% RSLogix 500 project SERVO_PROJECT.RSS, saved by version 8.30.00.16 %
PROJECT "UNTITLED"    % processor: Bul.1763 MicroLogix 1100 Series B %

PROGRAM FILES
  LAD 2 "MAIN"  4 rungs
  LAD 3 "INPUT"  7 rungs
  LAD 4 "OUTPUT"  2 rungs
  LAD 5 "CONTROL"  29 rungs

DATA FILES
  O0 OUTPUT  4 elements
  I1 INPUT  6 elements
  S2 STATUS  66 elements
  B3 BINARY  4 elements
  T4 TIMER  3 elements
  C5 COUNTER  1 elements
  R6 CONTROL  1 elements
  N7 INTEGER  4 elements
  F8 FLOAT  1 elements

LADDER 2 "MAIN"
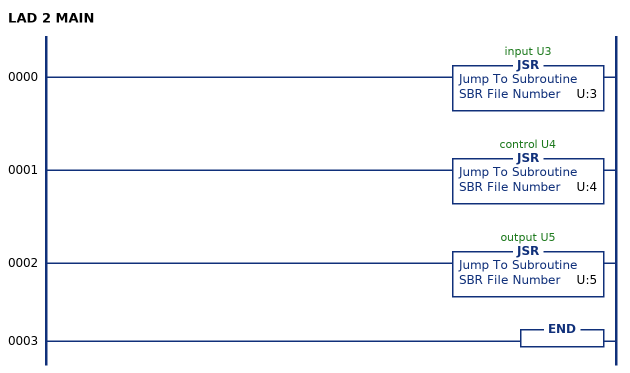
% Rung: 0 %
SOR JSR U:3 EOR
%   U:3  U3  "input" %
% Rung: 1 %
SOR JSR U:4 EOR
%   U:4  U4  "control" %
% Rung: 2 %
SOR JSR U:5 EOR
%   U:5  U5  "output" %
% Rung: 3 %
SOR END EOR

LADDER 3 "INPUT"
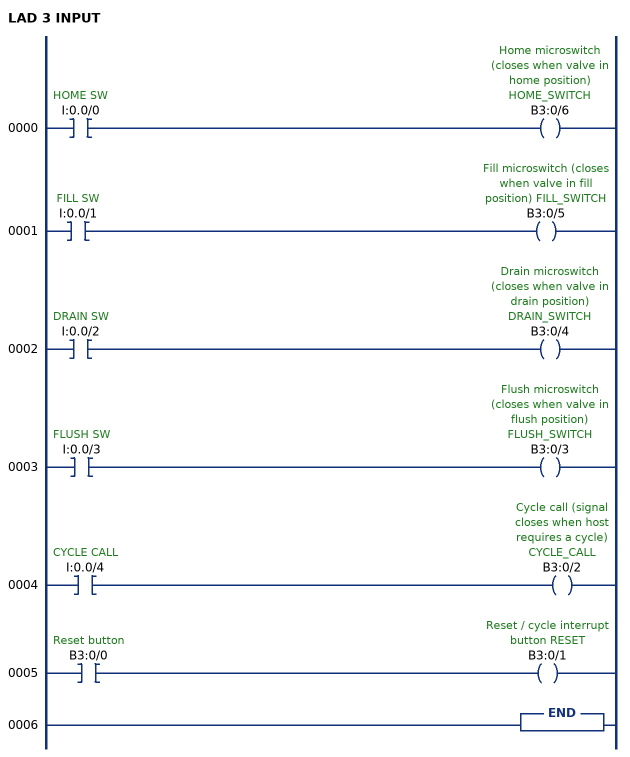
% Rung: 0 %
SOR XIC I:0.0/0 OTE B3:0/6 EOR
%   I:0.0/0  "HOME SW" %
%   B3:0/6  HOME_SWITCH  "Home microswitch (closes when valve in home position)" %
% Rung: 1 %
SOR XIC I:0.0/1 OTE B3:0/5 EOR
%   I:0.0/1  "FILL SW" %
%   B3:0/5  FILL_SWITCH  "Fill microswitch (closes when valve in fill position)" %
% Rung: 2 %
SOR XIC I:0.0/2 OTE B3:0/4 EOR
%   I:0.0/2  "DRAIN SW" %
%   B3:0/4  DRAIN_SWITCH  "Drain microswitch (closes when valve in drain position)" %
% Rung: 3 %
SOR XIC I:0.0/3 OTE B3:0/3 EOR
%   I:0.0/3  "FLUSH SW" %
%   B3:0/3  FLUSH_SWITCH  "Flush microswitch (closes when valve in flush position)" %
% Rung: 4 %
SOR XIC I:0.0/4 OTE B3:0/2 EOR
%   I:0.0/4  "CYCLE CALL" %
%   B3:0/2  CYCLE_CALL  "Cycle call (signal closes when host requires a cycle)" %
% Rung: 5 %
SOR XIC B3:0/0 OTE B3:0/1 EOR
%   B3:0/0  "Reset button" %
%   B3:0/1  RESET  "Reset / cycle interrupt button" %
% Rung: 6 %
SOR END EOR

LADDER 4 "OUTPUT"
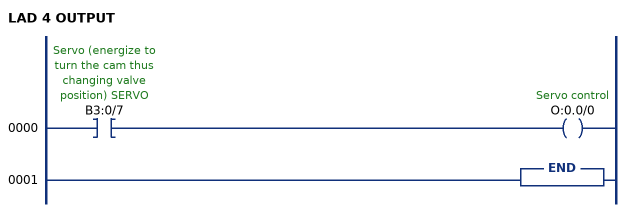
% Rung: 0 %
SOR XIC B3:0/7 OTE O:0.0/0 EOR
%   B3:0/7  SERVO  "Servo (energize to turn the cam thus changing valve position)" %
%   O:0.0/0  "Servo control" %
% Rung: 1 %
SOR END EOR

LADDER 5 "CONTROL"
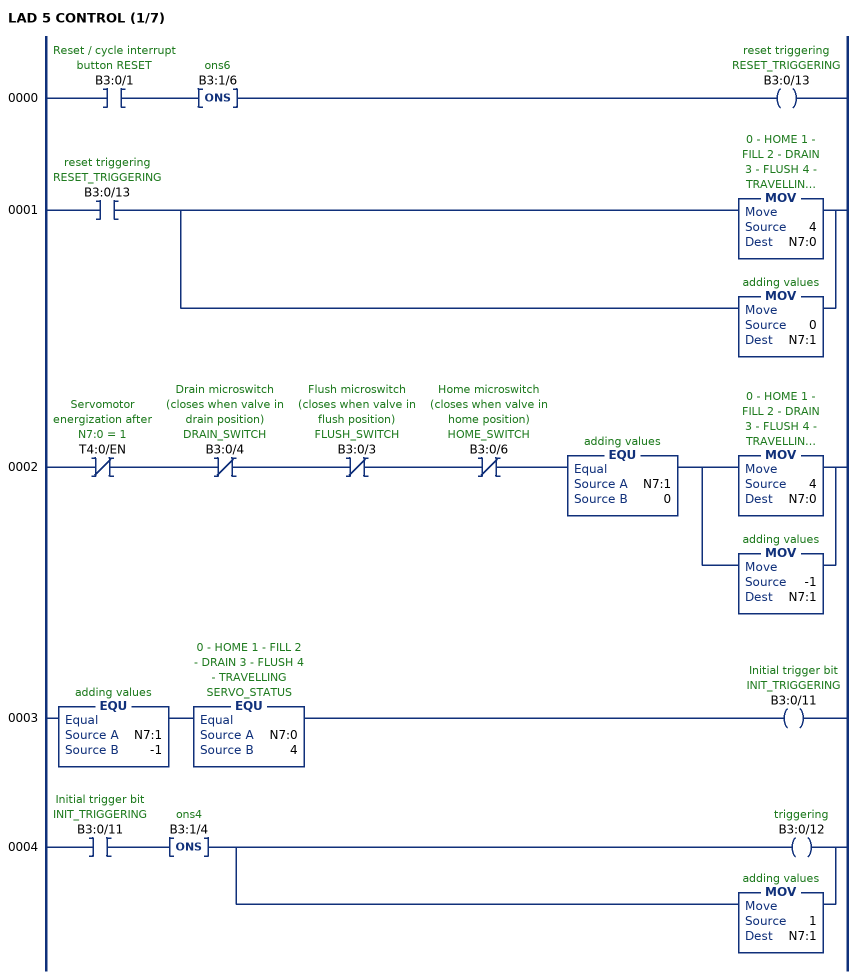
% Rung: 0 %
SOR XIC B3:0/1 ONS B3:1/6 OTE B3:0/13 EOR
%   B3:0/1  RESET  "Reset / cycle interrupt button" %
%   B3:1/6  "ons6" %
%   B3:0/13  RESET_TRIGGERING  "reset triggering" %
% Rung: 1 %
SOR XIC B3:0/13 BST MOV 4 N7:0 NXB MOV 0 N7:1 BND EOR
%   B3:0/13  RESET_TRIGGERING  "reset triggering" %
%   N7:0  SERVO_STATUS  "0 - HOME 1 - FILL 2 - DRAIN 3 - FLUSH 4 - TRAVELLING" %
%   N7:1  "adding values" %
% Rung: 2 %
SOR XIO T4:0/EN XIO B3:0/4 XIO B3:0/3 XIO B3:0/6 EQU N7:1 0 BST MOV 4 N7:0 NXB MOV -1 N7:1 BND EOR
%   T4:0/EN  "Servomotor energization after N7:0 = 1" %
%   B3:0/4  DRAIN_SWITCH  "Drain microswitch (closes when valve in drain position)" %
%   B3:0/3  FLUSH_SWITCH  "Flush microswitch (closes when valve in flush position)" %
%   B3:0/6  HOME_SWITCH  "Home microswitch (closes when valve in home position)" %
%   N7:1  "adding values" %
%   N7:0  SERVO_STATUS  "0 - HOME 1 - FILL 2 - DRAIN 3 - FLUSH 4 - TRAVELLING" %
% Rung: 3 %
SOR EQU N7:1 -1 EQU N7:0 4 OTE B3:0/11 EOR
%   N7:1  "adding values" %
%   N7:0  SERVO_STATUS  "0 - HOME 1 - FILL 2 - DRAIN 3 - FLUSH 4 - TRAVELLING" %
%   B3:0/11  INIT_TRIGGERING  "Initial trigger bit" %
% Rung: 4 %
SOR XIC B3:0/11 ONS B3:1/4 BST OTE B3:0/12 NXB MOV 1 N7:1 BND EOR
%   B3:0/11  INIT_TRIGGERING  "Initial trigger bit" %
%   B3:1/4  "ons4" %
%   B3:0/12  "triggering" %
%   N7:1  "adding values" %

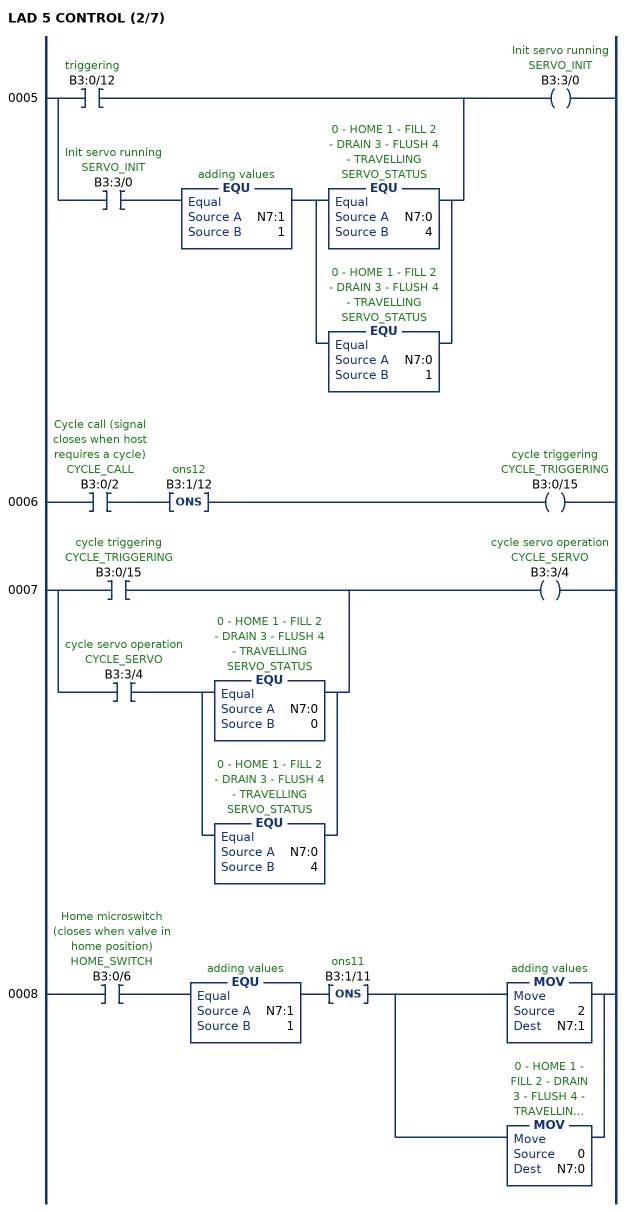
% Rung: 5 %
SOR BST XIC B3:0/12 NXB XIC B3:3/0 EQU N7:1 1 BST EQU N7:0 4 NXB EQU N7:0 1 BND BND OTE B3:3/0 EOR
%   B3:0/12  "triggering" %
%   B3:3/0  SERVO_INIT  "Init servo running" %
%   N7:1  "adding values" %
%   N7:0  SERVO_STATUS  "0 - HOME 1 - FILL 2 - DRAIN 3 - FLUSH 4 - TRAVELLING" %
% Rung: 6 %
SOR XIC B3:0/2 ONS B3:1/12 OTE B3:0/15 EOR
%   B3:0/2  CYCLE_CALL  "Cycle call (signal closes when host requires a cycle)" %
%   B3:1/12  "ons12" %
%   B3:0/15  CYCLE_TRIGGERING  "cycle triggering" %
% Rung: 7 %
SOR BST XIC B3:0/15 NXB XIC B3:3/4 BST EQU N7:0 0 NXB EQU N7:0 4 BND BND OTE B3:3/4 EOR
%   B3:0/15  CYCLE_TRIGGERING  "cycle triggering" %
%   B3:3/4  CYCLE_SERVO  "cycle servo operation" %
%   N7:0  SERVO_STATUS  "0 - HOME 1 - FILL 2 - DRAIN 3 - FLUSH 4 - TRAVELLING" %
% Rung: 8 %
SOR XIC B3:0/6 EQU N7:1 1 ONS B3:1/11 BST MOV 2 N7:1 NXB MOV 0 N7:0 BND EOR
%   B3:0/6  HOME_SWITCH  "Home microswitch (closes when valve in home position)" %
%   N7:1  "adding values" %
%   B3:1/11  "ons11" %
%   N7:0  SERVO_STATUS  "0 - HOME 1 - FILL 2 - DRAIN 3 - FLUSH 4 - TRAVELLING" %

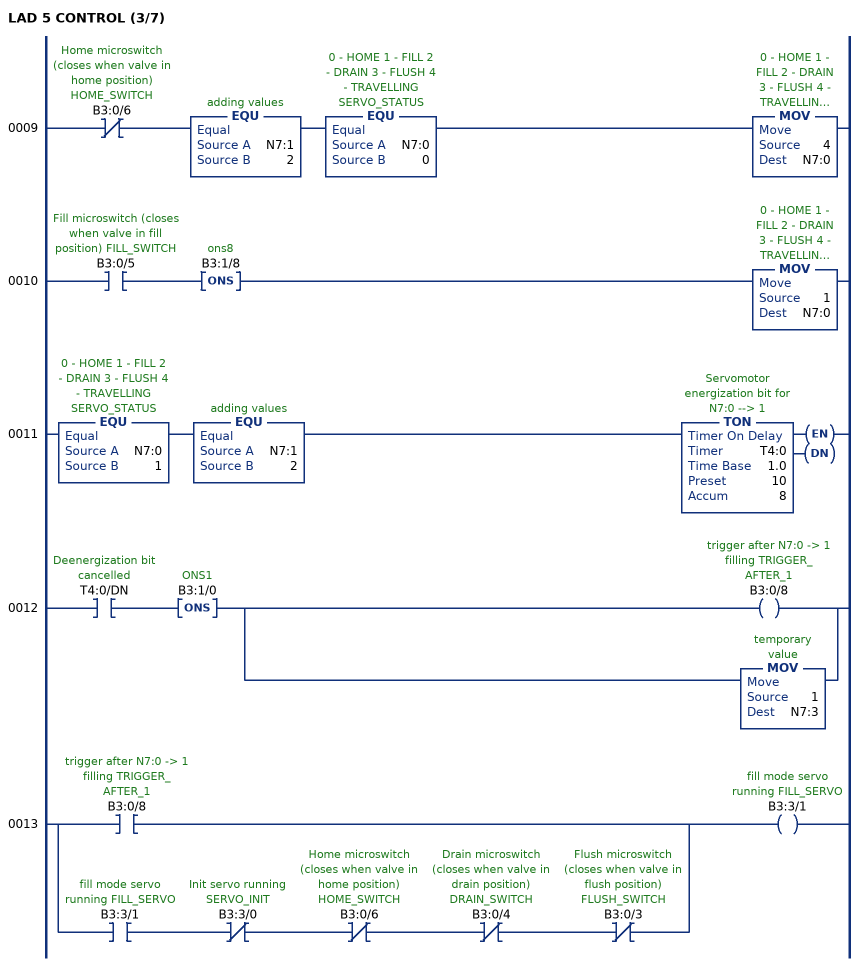
% Rung: 9 %
SOR XIO B3:0/6 EQU N7:1 2 EQU N7:0 0 MOV 4 N7:0 EOR
%   B3:0/6  HOME_SWITCH  "Home microswitch (closes when valve in home position)" %
%   N7:1  "adding values" %
%   N7:0  SERVO_STATUS  "0 - HOME 1 - FILL 2 - DRAIN 3 - FLUSH 4 - TRAVELLING" %
% Rung: 10 %
SOR XIC B3:0/5 ONS B3:1/8 MOV 1 N7:0 EOR
%   B3:0/5  FILL_SWITCH  "Fill microswitch (closes when valve in fill position)" %
%   B3:1/8  "ons8" %
%   N7:0  SERVO_STATUS  "0 - HOME 1 - FILL 2 - DRAIN 3 - FLUSH 4 - TRAVELLING" %
% Rung: 11 %
SOR EQU N7:0 1 EQU N7:1 2 TON T4:0 1.0 10 8 EOR
%   N7:0  SERVO_STATUS  "0 - HOME 1 - FILL 2 - DRAIN 3 - FLUSH 4 - TRAVELLING" %
%   N7:1  "adding values" %
%   T4:0  "Servomotor energization bit for N7:0 --> 1" %
% Rung: 12 %
SOR XIC T4:0/DN ONS B3:1/0 BST OTE B3:0/8 NXB MOV 1 N7:3 BND EOR
%   T4:0/DN  "Deenergization bit cancelled" %
%   B3:1/0  "ONS1" %
%   B3:0/8  TRIGGER_AFTER_1  "trigger after N7:0 -> 1 filling" %
%   N7:3  "temporary value" %
% Rung: 13 %
SOR BST XIC B3:0/8 NXB XIC B3:3/1 XIO B3:3/0 XIO B3:0/6 XIO B3:0/4 XIO B3:0/3 BND OTE B3:3/1 EOR
%   B3:0/8  TRIGGER_AFTER_1  "trigger after N7:0 -> 1 filling" %
%   B3:3/1  FILL_SERVO  "fill mode servo running" %
%   B3:3/0  SERVO_INIT  "Init servo running" %
%   B3:0/6  HOME_SWITCH  "Home microswitch (closes when valve in home position)" %
%   B3:0/4  DRAIN_SWITCH  "Drain microswitch (closes when valve in drain position)" %
%   B3:0/3  FLUSH_SWITCH  "Flush microswitch (closes when valve in flush position)" %

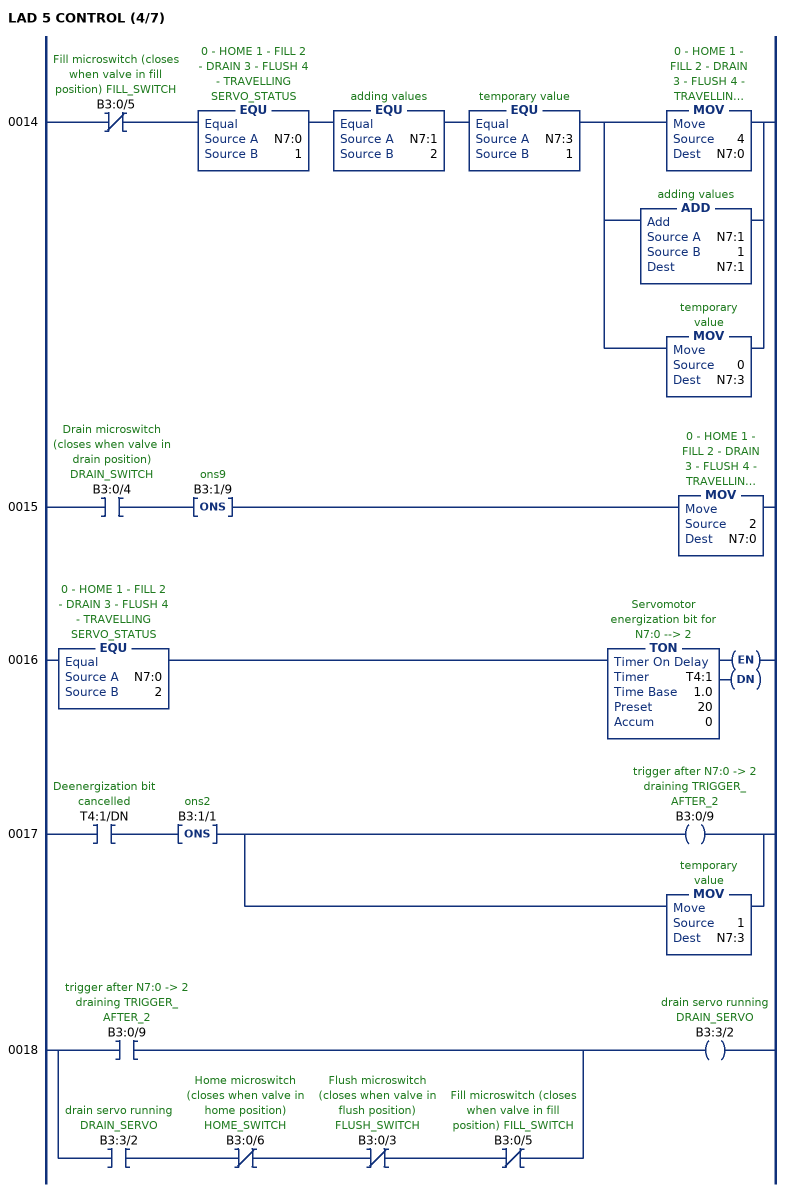
% Rung: 14 %
SOR XIO B3:0/5 EQU N7:0 1 EQU N7:1 2 EQU N7:3 1 BST MOV 4 N7:0 NXB ADD N7:1 1 N7:1 NXB MOV 0 N7:3 BND EOR
%   B3:0/5  FILL_SWITCH  "Fill microswitch (closes when valve in fill position)" %
%   N7:0  SERVO_STATUS  "0 - HOME 1 - FILL 2 - DRAIN 3 - FLUSH 4 - TRAVELLING" %
%   N7:1  "adding values" %
%   N7:3  "temporary value" %
% Rung: 15 %
SOR XIC B3:0/4 ONS B3:1/9 MOV 2 N7:0 EOR
%   B3:0/4  DRAIN_SWITCH  "Drain microswitch (closes when valve in drain position)" %
%   B3:1/9  "ons9" %
%   N7:0  SERVO_STATUS  "0 - HOME 1 - FILL 2 - DRAIN 3 - FLUSH 4 - TRAVELLING" %
% Rung: 16 %
SOR EQU N7:0 2 TON T4:1 1.0 20 0 EOR
%   N7:0  SERVO_STATUS  "0 - HOME 1 - FILL 2 - DRAIN 3 - FLUSH 4 - TRAVELLING" %
%   T4:1  "Servomotor energization bit for N7:0 --> 2" %
% Rung: 17 %
SOR XIC T4:1/DN ONS B3:1/1 BST OTE B3:0/9 NXB MOV 1 N7:3 BND EOR
%   T4:1/DN  "Deenergization bit cancelled" %
%   B3:1/1  "ons2" %
%   B3:0/9  TRIGGER_AFTER_2  "trigger after N7:0 -> 2 draining" %
%   N7:3  "temporary value" %
% Rung: 18 %
SOR BST XIC B3:0/9 NXB XIC B3:3/2 XIO B3:0/6 XIO B3:0/3 XIO B3:0/5 BND OTE B3:3/2 EOR
%   B3:0/9  TRIGGER_AFTER_2  "trigger after N7:0 -> 2 draining" %
%   B3:3/2  DRAIN_SERVO  "drain servo running" %
%   B3:0/6  HOME_SWITCH  "Home microswitch (closes when valve in home position)" %
%   B3:0/3  FLUSH_SWITCH  "Flush microswitch (closes when valve in flush position)" %
%   B3:0/5  FILL_SWITCH  "Fill microswitch (closes when valve in fill position)" %

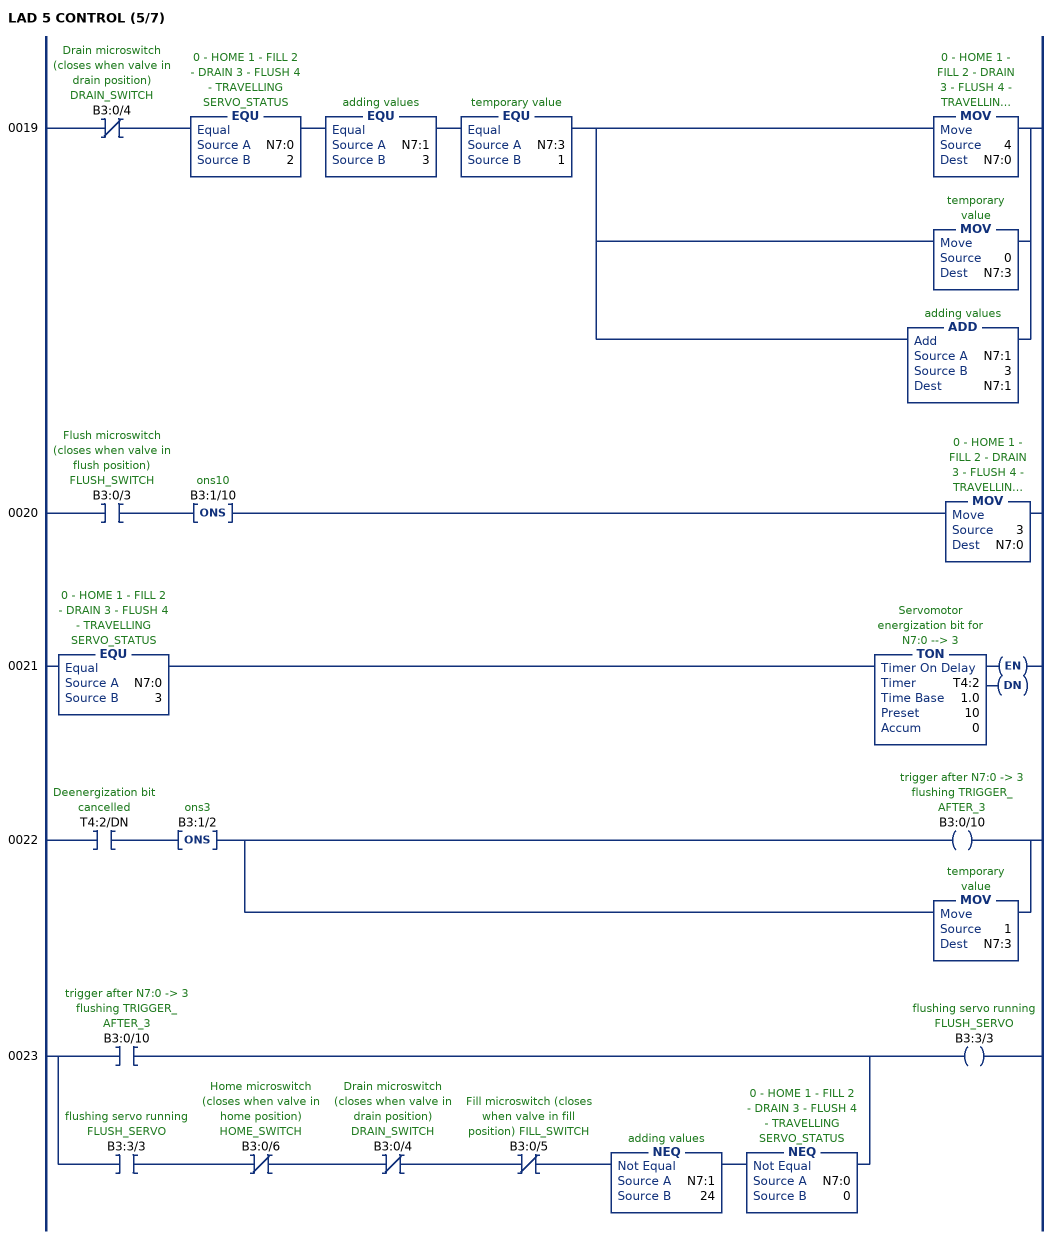
% Rung: 19 %
SOR XIO B3:0/4 EQU N7:0 2 EQU N7:1 3 EQU N7:3 1 BST MOV 4 N7:0 NXB MOV 0 N7:3 NXB ADD N7:1 3 N7:1 BND EOR
%   B3:0/4  DRAIN_SWITCH  "Drain microswitch (closes when valve in drain position)" %
%   N7:0  SERVO_STATUS  "0 - HOME 1 - FILL 2 - DRAIN 3 - FLUSH 4 - TRAVELLING" %
%   N7:1  "adding values" %
%   N7:3  "temporary value" %
% Rung: 20 %
SOR XIC B3:0/3 ONS B3:1/10 MOV 3 N7:0 EOR
%   B3:0/3  FLUSH_SWITCH  "Flush microswitch (closes when valve in flush position)" %
%   B3:1/10  "ons10" %
%   N7:0  SERVO_STATUS  "0 - HOME 1 - FILL 2 - DRAIN 3 - FLUSH 4 - TRAVELLING" %
% Rung: 21 %
SOR EQU N7:0 3 TON T4:2 1.0 10 0 EOR
%   N7:0  SERVO_STATUS  "0 - HOME 1 - FILL 2 - DRAIN 3 - FLUSH 4 - TRAVELLING" %
%   T4:2  "Servomotor energization bit for N7:0 --> 3" %
% Rung: 22 %
SOR XIC T4:2/DN ONS B3:1/2 BST OTE B3:0/10 NXB MOV 1 N7:3 BND EOR
%   T4:2/DN  "Deenergization bit cancelled" %
%   B3:1/2  "ons3" %
%   B3:0/10  TRIGGER_AFTER_3  "trigger after N7:0 -> 3 flushing" %
%   N7:3  "temporary value" %
% Rung: 23 %
SOR BST XIC B3:0/10 NXB XIC B3:3/3 XIO B3:0/6 XIO B3:0/4 XIO B3:0/5 NEQ N7:1 24 NEQ N7:0 0 BND OTE B3:3/3 EOR
%   B3:0/10  TRIGGER_AFTER_3  "trigger after N7:0 -> 3 flushing" %
%   B3:3/3  FLUSH_SERVO  "flushing servo running" %
%   B3:0/6  HOME_SWITCH  "Home microswitch (closes when valve in home position)" %
%   B3:0/4  DRAIN_SWITCH  "Drain microswitch (closes when valve in drain position)" %
%   B3:0/5  FILL_SWITCH  "Fill microswitch (closes when valve in fill position)" %
%   N7:1  "adding values" %
%   N7:0  SERVO_STATUS  "0 - HOME 1 - FILL 2 - DRAIN 3 - FLUSH 4 - TRAVELLING" %

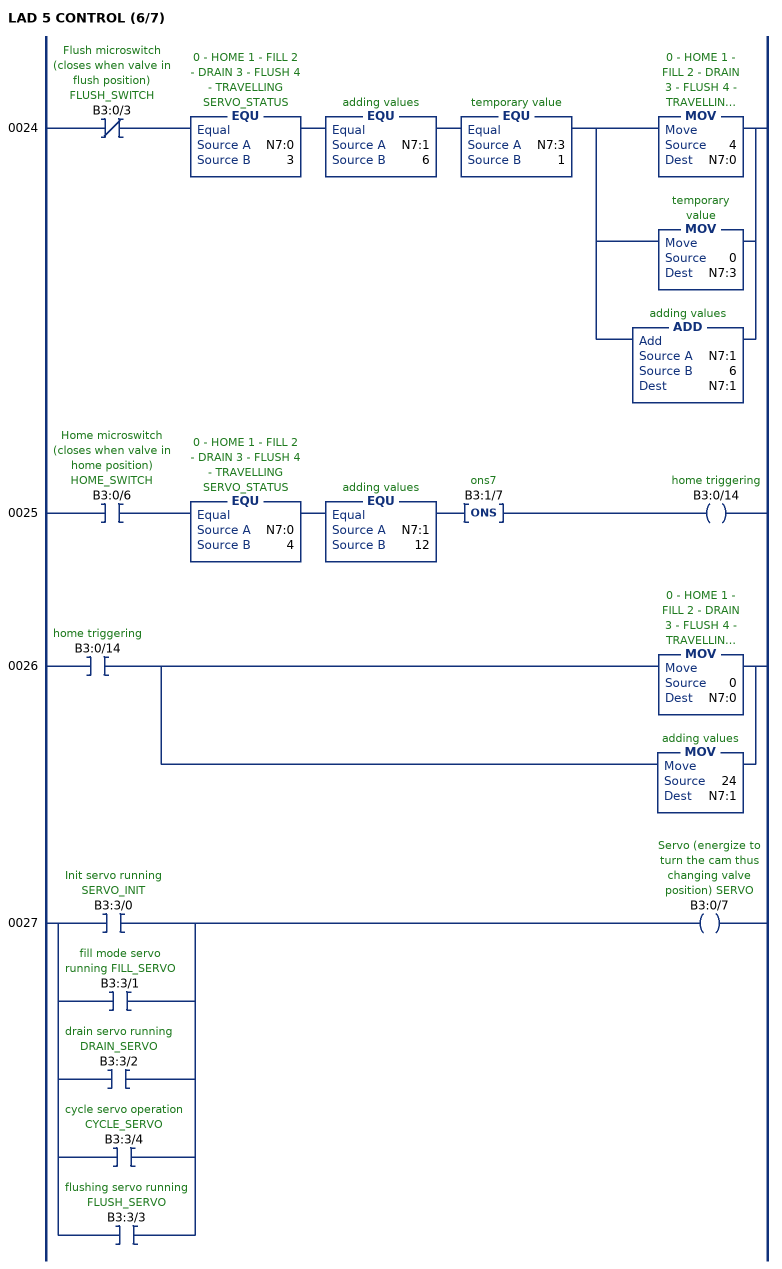
% Rung: 24 %
SOR XIO B3:0/3 EQU N7:0 3 EQU N7:1 6 EQU N7:3 1 BST MOV 4 N7:0 NXB MOV 0 N7:3 NXB ADD N7:1 6 N7:1 BND EOR
%   B3:0/3  FLUSH_SWITCH  "Flush microswitch (closes when valve in flush position)" %
%   N7:0  SERVO_STATUS  "0 - HOME 1 - FILL 2 - DRAIN 3 - FLUSH 4 - TRAVELLING" %
%   N7:1  "adding values" %
%   N7:3  "temporary value" %
% Rung: 25 %
SOR XIC B3:0/6 EQU N7:0 4 EQU N7:1 12 ONS B3:1/7 OTE B3:0/14 EOR
%   B3:0/6  HOME_SWITCH  "Home microswitch (closes when valve in home position)" %
%   N7:0  SERVO_STATUS  "0 - HOME 1 - FILL 2 - DRAIN 3 - FLUSH 4 - TRAVELLING" %
%   N7:1  "adding values" %
%   B3:1/7  "ons7" %
%   B3:0/14  "home triggering" %
% Rung: 26 %
SOR XIC B3:0/14 BST MOV 0 N7:0 NXB MOV 24 N7:1 BND EOR
%   B3:0/14  "home triggering" %
%   N7:0  SERVO_STATUS  "0 - HOME 1 - FILL 2 - DRAIN 3 - FLUSH 4 - TRAVELLING" %
%   N7:1  "adding values" %
% Rung: 27 %
SOR BST XIC B3:3/0 NXB XIC B3:3/1 NXB XIC B3:3/2 NXB XIC B3:3/4 NXB XIC B3:3/3 BND OTE B3:0/7 EOR
%   B3:3/0  SERVO_INIT  "Init servo running" %
%   B3:3/1  FILL_SERVO  "fill mode servo running" %
%   B3:3/2  DRAIN_SERVO  "drain servo running" %
%   B3:3/4  CYCLE_SERVO  "cycle servo operation" %
%   B3:3/3  FLUSH_SERVO  "flushing servo running" %
%   B3:0/7  SERVO  "Servo (energize to turn the cam thus changing valve position)" %

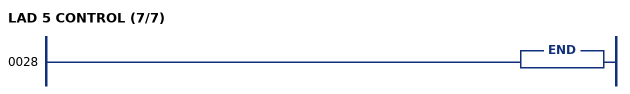
% Rung: 28 %
SOR END EOR

OTHER DOCUMENTED ADDRESSES
  B3:1/5  "ons5"

DATA TABLE (non-zero values as saved)
DATA T4
% .PRE .ACC %
% T4:0 % 10 8
% T4:1 % 20 0
% T4:2 % 10 0
